(* PLC project Unnamed, Unknown Unnamed 1 *)
(* stored: creationDateTime 2022-10-16T10:53:06, modificationDateTime 2023-09-26T20:34:45 *)

PROGRAM Actuators
  VAR
    OPTO_00 AT %IX0.0 : BOOL;  (* Stack 0 Opto Input 0 *)
    OPTO_01 AT %IX0.1 : BOOL;  (* Stack 0 Opto Input 1 *)
    OPTO_02 AT %IX0.2 : BOOL;  (* Stack 0 Opto Input 2 *)
    OPTO_03 AT %IX0.3 : BOOL;  (* Stack 0 Opto Input 3 *)
    OPTO_04 AT %IX0.4 : BOOL;  (* Stack 0 Opto Input 4 *)
    OPTO_05 AT %IX0.5 : BOOL;  (* Stack 0 Opto Input 5 *)
    OPTO_06 AT %IX0.6 : BOOL;  (* Stack 0 Opto Input 6 *)
    OPTO_07 AT %IX0.7 : BOOL;  (* Stack 0 Opto Input 7 *)
    OPTO_10 AT %IX1.0 : BOOL;  (* Stack 1 Opto Input 0 *)
    OPTO_11 AT %IX1.1 : BOOL;  (* Stack 1 Opto Input 1 *)
    OPTO_12 AT %IX1.2 : BOOL;  (* Stack 1 Opto Input 2 *)
    OPTO_13 AT %IX1.3 : BOOL;  (* Stack 1 Opto Input 3 *)
    OPTO_14 AT %IX1.4 : BOOL;  (* Stack 1 Opto Input 4 *)
    OPTO_15 AT %IX1.5 : BOOL;  (* Stack 1 Opto Input 5 *)
    OPTO_16 AT %IX1.6 : BOOL;  (* Stack 1 Opto Input 6 *)
    OPTO_17 AT %IX1.7 : BOOL;  (* Stack 1 Opto Input 7 *)
    RELAY_00 AT %QX0.0 : BOOL;  (* Stack 0 Relay 0 *)
    RELAY_01 AT %QX0.1 : BOOL;  (* Stack 0 Relay 1 *)
    RELAY_02 AT %QX0.2 : BOOL;  (* Stack 0 Relay 2 *)
    RELAY_03 AT %QX0.3 : BOOL;  (* Stack 0 Relay 3 *)
    RELAY_04 AT %QX0.4 : BOOL;  (* Stack 0 Relay 4 *)
    RELAY_05 AT %QX0.5 : BOOL;  (* Stack 0 Relay 5 *)
    RELAY_06 AT %QX0.6 : BOOL;  (* Stack 0 Relay 6 *)
    RELAY_07 AT %QX0.7 : BOOL;  (* Stack 0 Relay 7 *)
    RELAY_10 AT %QX1.0 : BOOL;  (* Stack 1 Relay 0 *)
    RELAY_11 AT %QX1.1 : BOOL;  (* Stack 1 Relay 1 *)
    RELAY_12 AT %QX1.2 : BOOL;  (* Stack 1 Relay 2 *)
    RELAY_13 AT %QX1.3 : BOOL;  (* Stack 1 Relay 3 *)
    RELAY_14 AT %QX1.4 : BOOL;  (* Stack 1 Relay 4 *)
    RELAY_15 AT %QX1.5 : BOOL;  (* Stack 1 Relay 5 *)
    RELAY_16 AT %QX1.6 : BOOL;  (* Stack 1 Relay 6 *)
    RELAY_17 AT %QX1.7 : BOOL;  (* Stack 1 Relay 7 *)
  END_VAR

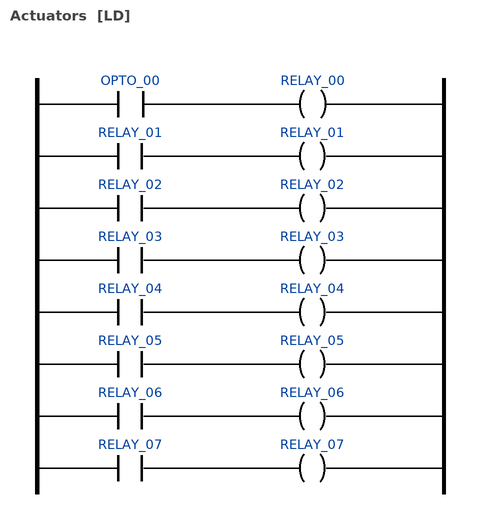
(* LD diagram, written out as Structured Text *)
RELAY_00 := OPTO_00;
RELAY_01 := RELAY_01;
RELAY_02 := RELAY_02;
RELAY_03 := RELAY_03;
RELAY_04 := RELAY_04;
RELAY_05 := RELAY_05;
RELAY_06 := RELAY_06;
RELAY_07 := RELAY_07;
END_PROGRAM

CONFIGURATION Config0
  RESOURCE Res0 ON PLC
    TASK task0(INTERVAL := T#20ms, PRIORITY := 0);
    PROGRAM instance0 WITH task0 : Actuators;
  END_RESOURCE
END_CONFIGURATION
